TYPE ST_Powermodule_PowerCurveCoefficients :
STRUCT
	enable: BOOL;
	a : REAL;
	b : REAL;
	c : REAL;
	d : REAL; 
	e : REAL;
	f : REAL;
END_STRUCT
END_TYPE

(* stored: Version 1.1.0.1, ProductVersion 3.1.4026.18
   DUT ST_Powermodule_PowerCurveCoefficients: Id {372a3234-6cd0-4ad6-b245-ea889a630a1a} *)
